{attribute 'hide'}
TYPE St_Error :
STRUCT
	
END_STRUCT
END_TYPE

(* stored: Version 1.1.0.1, ProductVersion 3.1.4024.6
   DUT St_Error: Id {9b006677-b501-446d-a72a-96a3d8d20e34} *)
